ADAPTER A2X2 (* bidirectional Adapter Interface for 2 Events and 2 Bools *)
  (* Standard: 61499-1; Description: Copyright (c) 2026 HR Agrartechnik GmbH This program and the accompanying materials are made available under the terms of the Eclipse Public License 2.0 which is available at https://www.eclipse.org/legal/epl-2.0/ SPDX-License-Identifier: EPL-2.0 *)
  (* Version 1.0, 2026-08-31, Franz Höpfinger, HR Agrartechnik GmbH, Initial Version *)
  PACKAGE adapter::types::bidirectional;
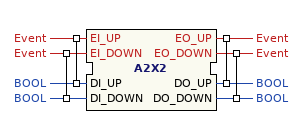
  EVENT_INPUT
    EI_UP WITH DI_UP; (* UP Request (or Indication) *)
    EI_DOWN WITH DI_DOWN; (* DOWN Request (or Indication) *)
  END_EVENT
  EVENT_OUTPUT
    EO_UP WITH DO_UP; (* UP Indication (or Request) *)
    EO_DOWN WITH DO_DOWN; (* DOWN Indication (or Request) *)
  END_EVENT
  VAR_INPUT
    DI_UP : BOOL; (* TRUE = forward, up, right, clockwise *)
    DI_DOWN : BOOL; (* TRUE = backward, down, left, counter-clockwise *)
  END_VAR
  VAR_OUTPUT
    DO_UP : BOOL; (* TRUE = forward, up, right, clockwise *)
    DO_DOWN : BOOL; (* TRUE = backward, down, left, counter-clockwise *)
  END_VAR
END_ADAPTER
